DATA_BLOCK "MotorData"
VAR
  Ton : Array[0..50] of TON_TIME;
  P : Array[0..50] of Bool;
  Time : Array[0..50] of Time;
END_VAR
BEGIN
END_DATA_BLOCK
